TYPE ST_Module :
STRUCT
	CloseChargeRly	: BOOL;
	OpenDumpRly		: BOOL;
	Fire			: BOOL;
	TriggerScope	: BOOL;
	
	ChargeRly_close	: BOOL;
	DumpRly_open	: BOOL;
	ModuleCharged	: BOOL;
	VoltageFeedback : DINT;
END_STRUCT
END_TYPE

(* stored: Version 1.1.0.1, ProductVersion 3.1.4024.11
   DUT ST_Module: Id {dc37cb22-2b59-4e70-80e4-3268cd948482} *)
